PROGRAM MAIN
VAR
	bStartExport : BOOL;
	bStartImport : BOOL;
	bStartAquisition : BOOL;

END_VAR

IF bStartExport THEN
	bStartExport := FALSE;
	DBSync(bExportTrigger := TRUE);
ELSIF bStartImport THEN
	bStartImport := FALSE;
	DBSync(bImportTrigger := TRUE);
ELSIF bStartAquisition THEN
	pTimer();
END_IF

END_PROGRAM

(* stored: Version 1.1.0.1, ProductVersion 3.1.4024.12
   POU MAIN: Id {9ad4ba43-e79f-4762-b016-8ed016718c25}, SpecialFunc None *)
